{attribute addProperty BoxType "EL2595-0000-0019"}
{attribute addProperty Id "Ready_to_activateBIT10.1251Output_activeBIT10.1252Switching_operation_counter_BIT_0BIT10.1254Switching_operation_counter_BIT_1BIT10.1254Switching_operation_counter_BIT_2BIT10.1254WarningBIT10.1257ErrorBIT10.1258Digital_inputBIT10.12512TxPDO_ToggleBIT10.12516"}
{attribute addProperty CRC "558331878"}
{attribute addProperty SizeInBites "16"}
{attribute addProperty SizeInBytes "2"}
TYPE Status_214777E6 :
STRUCT
	{attribute addProperty Name "Ready_to_activate"}
	Ready_to_activate : BIT;
	{attribute addProperty Name "Output_active"}
	Output_active : BIT;
	{attribute 'hide'}
	reserve_1 : BIT;
	{attribute addProperty Name "Switching_operation_counter"}
	Switching_operation_counter_BIT_0 : BIT;
	{attribute addProperty Name "Switching_operation_counter"}
	Switching_operation_counter_BIT_1 : BIT;
	{attribute addProperty Name "Switching_operation_counter"}
	Switching_operation_counter_BIT_2 : BIT;
	{attribute addProperty Name "Warning"}
	Warning : BIT;
	{attribute addProperty Name "Error"}
	Error : BIT;
	{attribute 'hide'}
	reserve_2_BIT_0 : BIT;
	{attribute 'hide'}
	reserve_2_BIT_1 : BIT;
	{attribute 'hide'}
	reserve_2_BIT_2 : BIT;
	{attribute addProperty Name "Digital_input"}
	Digital_input : BIT;
	{attribute 'hide'}
	reserve_3_BIT_0 : BIT;
	{attribute 'hide'}
	reserve_3_BIT_1 : BIT;
	{attribute 'hide'}
	reserve_3_BIT_2 : BIT;
	{attribute addProperty Name "TxPDO_Toggle"}
	TxPDO_Toggle : BIT;
END_STRUCT
END_TYPE

(* stored: Version 1.2.0.0, ProductVersion 3.1.4024.9
   DUT Status_214777E6: Id {12371112-7796-4d7d-b9b6-5cc5633ccecd} *)
